// TIA Portal V19 export
DATA_BLOCK "DI_FW_POS_1"   // DB21
// stored: AutoNumber false, InstanceOfName FB_POS_FW_INC, InstanceOfType FB
"FB_POS_FW_INC"
   // VAR_INPUT
   //    SysTime : Time := T#35M_13S_884MS;
   // END_VAR
   // VAR RETAIN
   //    Config : Struct
   //       Speed : Struct
   //          Min : Int := 5;
   //          Tipp : Int := 10;
   //          Hand : Int := 50;
   //          Max : Int := 100;
   //          Norm : Real := 800.0;
   //          endMess : Real := 800.4667;
   //       END_STRUCT;
   //       Rampe : Struct
   //          Auf_Leer : Real := 3.0;
   //          Ab_Leer : Real := 3.0;
   //          Auf_Ware : Real := 5.0;
   //          Ab_Ware : Real := 5.0;
   //          NotStop : Real := 1.0;
   //       END_STRUCT;
   //       Bereich : Struct
   //          Pos : DInt := 10;
   //          Stop : DInt := 2;
   //          Ziel : DInt := 5;
   //          Schleich : DInt := 200;
   //          Langsam : DInt := 0;
   //       END_STRUCT;
   //       TV_Position : DInt := 1000;
   //       Reaktionszeit : Int := 50;
   //       Startzeit : Int := 200;
   //       Variante : Byte := 16#00;
   //       SimIstSpeed : Byte := 16#00;
   //       PlateauZeit : Int := 250;
   //    END_STRUCT;
   //    IN : Struct
   //       BA_Tipp : Bool := FALSE;
   //       BA_Hand : Bool := TRUE;
   //       BA_Auto : Bool := FALSE;
   //       LeerFahrt : Bool := TRUE;
   //       Frg_Fahren : Bool := FALSE;
   //       Frg_Eil : Bool := FALSE;
   //       Break_on : Bool := TRUE;
   //       res_2 : Bool := FALSE;
   //       resB : Byte := 16#00;
   //       PosInc : DInt := 1998;
   //       ZielInc : DInt := 0;
   //       IstSpeed : Int := 0;
   //    END_STRUCT;
   //    OUT : Struct
   //       Pos_ok : Bool := TRUE;
   //       Break_off : Bool := FALSE;
   //       res_1 : Bool := FALSE;
   //       res_2 : Bool := FALSE;
   //       res_3 : Bool := FALSE;
   //       res_4 : Bool := FALSE;
   //       res_5 : Bool := FALSE;
   //       res_6 : Bool := FALSE;
   //       resB : Byte := 16#00;
   //       Bereich_langsam : DInt := 0;
   //       SollSpeed : Int := 0;
   //    END_STRUCT;
   //    Tmp : Struct
   //       lastTime : DInt := 2113884;
   //       DiffTime : Real := 31.0;
   //       lastSpeed : Real := 0.0;
   //       Messung : Struct
   //          lastInc : Real := 1998.0;
   //          addInc : Real := 0.0;
   //          addTime : Real := 0.0;
   //          lastIst : Int := 0;
   //          messAct : Bool := FALSE;
   //       END_STRUCT;
   //       StopCount : DInt := 1_147_715_584;
   //       subInc : Real := 0.0;
   //       lastOut : Real := 0.0;
   //       TaktCount : Real := 0.0;
   //       RunTime : DInt := 0;
   //    END_STRUCT;
   // END_VAR
BEGIN
END_DATA_BLOCK
